{attribute addProperty BoxType "EL3423-0000-0016"}
{attribute addProperty Id "Reactive_EnergyAT %I*LINT64818Reactive_Positive_EnergyAT %I*ULINT64819Reactive_Negative_EnergyAT %I*ULINT64820"}
{attribute addProperty CRC "4165191566"}
{attribute addProperty SizeInBites "192"}
{attribute addProperty SizeInBytes "24"}
TYPE Total_Reactive_F843C78E :
STRUCT
	{attribute addProperty Name "Reactive_Energy"}
	Reactive_Energy AT %I* : LINT;
	{attribute addProperty Name "Reactive_Positive_Energy"}
	Reactive_Positive_Energy AT %I* : ULINT;
	{attribute addProperty Name "Reactive_Negative_Energy"}
	Reactive_Negative_Energy AT %I* : ULINT;
END_STRUCT
END_TYPE

(* stored: Version 1.2.0.0, ProductVersion 3.1.4024.9
   DUT Total_Reactive_F843C78E: Id {9355b6f8-1616-40e3-b692-131cb45030ef} *)
